{attribute 'linkalways'} 
{attribute 'no_explicit_call' := 'This FB is a CLASS and must be accessed using methods or properties'}
{attribute 'enable_dynamic_creation'}
FUNCTION_BLOCK FINAL ATAN_LREAL EXTENDS Node
VAR
	in : _LREAL(0.0);
	out : _LREAL(0.0);
END_VAR

METHOD PUBLIC Clone : I_Node
VAR
	pNode : POINTER TO ATAN_LREAL;
END_VAR
pNode := __NEW(ATAN_LREAL);
Clone := pNode^;
END_METHOD

METHOD FB_init : BOOL
VAR_INPUT
	bInitRetains : BOOL; // if TRUE, the retain variables are initialized (warm start / cold start)
	bInCopyCode : BOOL;  // if TRUE, the instance afterwards gets moved into the copy code (online change)
END_VAR
AddInput('in',THIS^.in);
AddOutput('out', THIS^.out);
END_METHOD

METHOD PROTECTED OnExecute
VAR
END_VAR
out.Value := ATAN(in.Value);
END_METHOD

END_FUNCTION_BLOCK

(* stored: Version 1.1.0.1, ProductVersion 3.1.4024.15
   POU ATAN_LREAL: Id {df27e399-46b8-4b5d-a75e-604515473952}, SpecialFunc None
   Folder Constructor: Id {51b9c3c4-ce05-443b-addf-d922171d5b80}
   Method Clone: Id {2a8d95d0-0c82-4a13-abb3-185602ce2f7b}
   Method FB_init: Id {99707a9e-157d-4524-bae1-1662f1f21f11}
   Method OnExecute: Id {e0823f90-af4f-4cb9-b83e-96ef572659ac} *)
